Fanuc KAREL source: IO0002.KL

-- PROVISIONAL review KL for V940-1; original PC SHA256 ac9eadbde8c8ae525fb3da3b4e5f21a2602c85e0d100375cda8be1233770324e
-- Incomplete behavior may be omitted. Consult companion uncertainty JSON. Do not deploy.
PROGRAM IO0002
%NOLOCKGROUP
-- UNRESOLVED_LOCAL_POOL 5 cells at code offset 13; source declarations unknown
-- DIRECT_LOCAL_WORD_ACCESS alone does not prove INTEGER, REAL, or BOOLEAN
BEGIN
  -- V9_EXPOSED_INDEXED_TABLE_HINT layout=0001; 1 counted words exposed once; source arms/runtime held
  -- V9_ZERO_GLOBAL_LAYOUT_HINT count-one $GROUP table, zero relocation slots, two routine descriptors; executable preamble and source held
  -- UNRESOLVED_PC offsets 0-18; opcodes 2B,2C,7B
  -- UNRESOLVED_PC offsets 23-30; opcodes 9D,23
  -- UNRESOLVED_PC offsets 35-49; opcodes 2E,22,9D,33,35
  -- UNRESOLVED_PC offsets 54-61; opcodes 9D,23
  -- UNRESOLVED_PC offsets 66-77; opcodes 2E,23
  -- UNRESOLVED_PC offsets 82-92; opcodes 9D,19,9D,57,79
  -- UNRESOLVED_PC offsets 97-111; opcodes 21,9D,52,23
  -- UNRESOLVED_PC offsets 121-125; opcodes 7F
  -- UNRESOLVED_PC offsets 130-134; opcodes 27,AA
  -- UNRESOLVED_PC offsets 139-143; opcodes 7F
END IO0002
